PROGRAM P_Demo_PULARGE_TO_ULARGE
VAR
    ulgRealValue           : ULARGE; // 模拟 wire 缓冲区中的 ULARGE 字段
    pULARGEField           : POINTER TO ULARGE; // 业务侧先算好的字段地址（ADR 或 pBase+nOff）
    bExtractField          : BOOL; // 在线置 TRUE 触发一次解析
    ulgRealValue_extracted : ULARGE; // 解析后的副本，供业务逻辑使用
END_VAR

// ============================================================
// Tc2_Utilities.PULARGE_TO_ULARGE 演示程序（FUNCTION）
// ============================================================
// 场景：从一段二进制 wire 缓冲区里按偏移取 ULARGE 字段（Modbus/CAN/ADS Raw）。
// 价值：替代手写 pField + nOff + ^ 指针算术；一次调用取值，少打错符号。
// 验证：在线写 ulgRealValue := 示例值；bExtractField := TRUE；
//       下一周期 ulgRealValue_extracted 应等于 ulgRealValue。
// ============================================================

// 业务代码通常已经算好字段地址（pBase + 协议偏移）；演示用 ADR 等价
pULARGEField := ADR(ulgRealValue);

IF bExtractField AND pULARGEField <> 0 THEN
    // 单次完整调用：避免手写 ^ 解引用，统一风格便于和字节序转换串联
    ulgRealValue_extracted := PULARGE_TO_ULARGE(pULARGEField);
    bExtractField := FALSE;
END_IF;

END_PROGRAM

(* stored: Version 1.1.0.1, ProductVersion 3.1.4024.5
   POU P_Demo_PULARGE_TO_ULARGE: Id {83beb941-06fc-5fcd-bd83-bc330418897d}, SpecialFunc None *)
